// TIA Portal V16 export
// export: Created 2022-11-17T11:55:36.8346482Z, ExportSetting WithDefaults, DisplayName Totally Integrated Automation Portal, DisplayVersion V16 Update 6, DisplayName TIA Portal Version Control Interface, DisplayVersion V16 Update 2, DisplayName TIA Portal Openness, DisplayVersion V16 Update 6, DisplayName SINAMICS Startdrive Advanced, DisplayVersion V16 Update 5, DisplayName SINAMICS Startdrive G130, G150, S120, S150, SINAMICS MV, S210, DisplayVersion V16 Update 5, DisplayName SINAMICS Startdrive G110M, G120, G120C, G120D, G120P, G115D, DisplayVersion V16 Update 5, DisplayName STEP 7 Professional, DisplayVersion V16 Update 6, DisplayName STEP 7 Safety, DisplayVersion V16, DisplayName WinCC Advanced, DisplayVersion V16 Update 6
DATA_BLOCK "DB322_APP"   // DB322
TITLE = PID
{ S7_Optimized_Access := 'FALSE' }
VERSION : 0.1
// stored: AutoNumber false, IsOnlyStoredInLoadMemory false, IsWriteProtectedInAS false
   VAR RETAIN
      IN0 : Int := 0;
      IN1 : Int := 0;
      IN2 : Int := 0;
      IN3 : Int := 0;
      IN4 : Int := 0;
      IN5 : Int := 0;
      IN6 : Int := 0;
      IN7 : Int := 0;
      IN8 : Int := 0;
      IN9 : Int := 0;
      IN10 : DInt := 224;
      IN11 : DInt := 240;
      IN12 : DInt := 0;   // TIRO EQUIVALENTE SU CELLA (kg)
      APP { S7_SetPoint := 'True'} : "APP";
   END_VAR
BEGIN
   APP.PID_ComponenteProporzionale := 0;
   APP.PID_ComponenteIntegrale := 0;
   APP.PID_ComponenteDerivativa := 0;
   APP.Tiro := 0;
   APP.Tiro1 := 0;
   APP.Tiro2 := 0;
   APP.TiroPrecedente := 0;
   APP.TiroAppoggio := 0;
   APP.ErroreAttuale := 0;
   APP.ErrorePrecedente := 0;
   APP.PID_Kp := 70;
   APP.PID_Ki := 60;
   APP.PID_Kd := 0;
   APP.SetpointTiro := 56;
   APP.SetpointTiroRampa := 750;
   APP.TransitorioInizialeFase1 := 0;
   APP.TransitorioFase3 := 1;
   APP.TransitorioFase4 := 1;
   APP.VelocitaRotazione := 5;
   APP.VelocitaRotazioneFase2 := 100;
   APP.VelocitaRotazioneAppoggio1 := 100;
   APP.VelocitaRotazioneAppoggio2 := 100;
   APP.Fase1OneShoot := 0;
   APP.Fase2OneShoot := 0;
   APP.Fase3OneShoot := 0;
   APP.Fase4OneShoot := 0;
   APP.ArrestoRepentinoOneShoot := 0;
   APP.TiroFase1 := 0;
   APP.TempIntero := 90;
   APP.Fase := 0;
   APP.BallerinoPrecedente[0..2] := 56;
   APP.LimiteComponenteIntegrale := 20000;
   APP.TiroRichiesto := 10;
   APP.TimerArrestoRepentino := 2;
   APP.TiroMinimoArrestoRepentino := 10;
   APP.VariazioneTiro := 0;
   APP.TimerFase2 := 0;
   APP.TempoRotturaFilm := 166;
   APP.TimerFase4 := 0;
   APP.TiroMinimoFase4 := 6;
   APP.PID_Uscita := 0;
   APP.PrestiroRichiesto := 300;
   APP.PrestiroAppoggio := 0.5;
END_DATA_BLOCK
